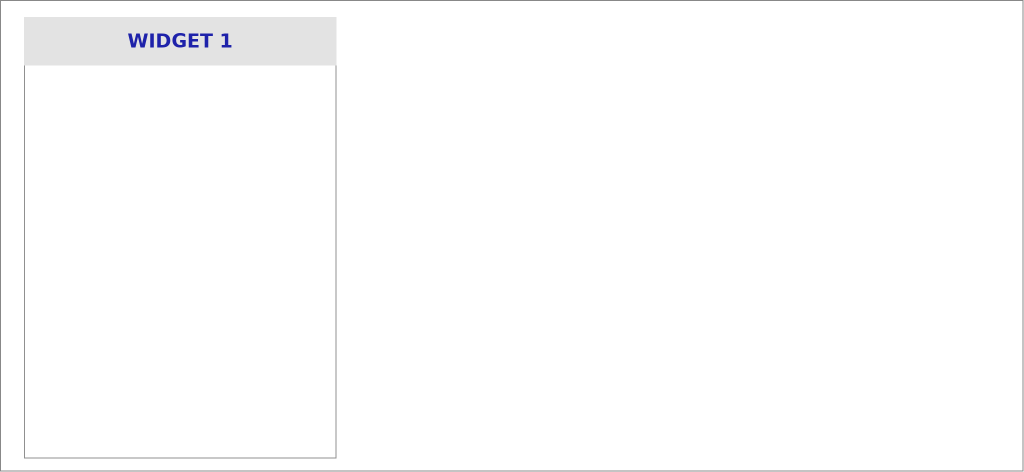
VISUALIZATION _001_Blank_1  // 1024x472
    GroupBox (24,16 312x442)
        Rectangle (0,1 312x48), "WIDGET 1"
END_VISUALIZATION

(* stored: Version 1.1.0.1, ProductVersion 3.1.4022.18
   Visu _001_Blank_1: Id {777d0601-9442-48d1-ac7f-a9c054590fdc} *)
